PROGRAM CONTAINER_TEST
VAR

    fbMotionLogger : FB_MotionLogger;
    // Persistant storage
    fbPersistentDataStorage : FB_PersistentDataStorage;
    fbMotionStage : FB_MotionStageNC(	sName := 'NC',
                                        AxisRef := NcAxis_GVL.NC,
                                        iMotionLogger := fbMotionLogger,
                                        iPersistentDataStorage := fbPersistentDataStorage
                                    );
END_VAR

fbMotionLogger();
fbPersistentDataStorage();
fbMotionStage();

END_PROGRAM

(* stored: Version 1.1.0.1
   POU CONTAINER_TEST: Id {cf068a0d-ba9f-4527-8e93-978663edefcc}, SpecialFunc None *)
